FUNCTION_BLOCK Reset5
VAR_INPUT
END_VAR
VAR_OUTPUT
END_VAR
VAR
END_VAR

END_FUNCTION_BLOCK

(* stored: Version 1.1.0.1, ProductVersion 3.1.4024.11
   POU Reset5: Id {d6eb2a38-1872-4524-ad8d-4a058018357e}, SpecialFunc None *)
